// TwinCAT 3 PLC project vgr
// ProgramVersion: 3.1.4023.0
// libraries:
//   Tc2_Standard, * (Beckhoff Automation GmbH)
//   Tc2_System, * (Beckhoff Automation GmbH)
//   Tc3_Module, * (Beckhoff Automation GmbH)
// project tree:
//   GVLs/ Encoder.TcGVL, Position.TcGVL, StartStop.TcGVL, VGR.TcGVL
//   / PlcTask.TcTTO
//   POUs/ AboutEqual.TcPOU, AxisMovementController.TcPOU, AxisReferencing.TcPOU, EncoderSignalProcessor.TcPOU, MAIN.TcPOU, AxisController.TcPOU, VGR_State.TcPOU
// real-time tasks:
//   TASK PlcTask: cycle T#10ms, priority 20, ADS port 350
// I/O:
//   DEVICE Device 1 (EtherCAT), AmsNetId 172.23.144.1.2.1
//     Term 1 (EK1100) [EK1100 EtherCAT Coupler (2A E-Bus)]
//       Term 2 (EL1809) [EL1809 16Ch. Dig. Input 24V, 3ms]
//       Term 3 (EL2809) [EL2809 16Ch. Dig. Output 24V, 0.5A]
//       Term 4 (EL2535-0002) [EL2535-0002 2Ch. Pulse Width Current Output (24V, 2 A)]
//       Term 5 (EL2535-0002) [EL2535-0002 2Ch. Pulse Width Current Output (24V, 2 A)]
//       Term 6 (EL5152) [EL5152 2Ch. Inc. Encoder]
//       Term 7 (EL5152) [EL5152 2Ch. Inc. Encoder]
//       Term 8 (EL9011) [EL9011 End Terminal]
// variable links:
//   vgr/vgr Instance <-> Device 1 (EtherCAT)/Term 1 (EK1100)/Term 2 (EL1809)
//     PlcTask Inputs/StartStop.IX_START <-> Channel 11/Input
//     PlcTask Inputs/StartStop.IX_STOP <-> Channel 10/Input
//     PlcTask Inputs/VGR.IX_VGR_RefSwitchHorizontalAxis_I2 <-> Channel 2/Input
//     PlcTask Inputs/VGR.IX_VGR_RefSwitchRotate_I3 <-> Channel 3/Input
//     PlcTask Inputs/VGR.IX_VGR_RefSwitchVerticalAxis_I1 <-> Channel 1/Input
//   vgr/vgr Instance <-> Device 1 (EtherCAT)/Term 1 (EK1100)/Term 3 (EL2809)
//     PlcTask Outputs/VGR.QX_VGR_Compressor_Q7 <-> Channel 7/Output
//     PlcTask Outputs/VGR.QX_VGR_M1_VerticalAxisDown_Q2 <-> Channel 2/Output
//     PlcTask Outputs/VGR.QX_VGR_M1_VerticalAxisUp_Q1 <-> Channel 1/Output
//     PlcTask Outputs/VGR.QX_VGR_M2_HorizontalAxisBackward_Q3 <-> Channel 3/Output
//     PlcTask Outputs/VGR.QX_VGR_M2_HorizontalAxisForward_Q4 <-> Channel 4/Output
//     PlcTask Outputs/VGR.QX_VGR_M3_RotateClockwise_Q5 <-> Channel 5/Output
//     PlcTask Outputs/VGR.QX_VGR_M3_RotateCounterclockwise_Q6 <-> Channel 6/Output
//     PlcTask Outputs/VGR.QX_VGR_ValveVacuum_Q8 <-> Channel 8/Output
//   vgr/vgr Instance <-> Device 1 (EtherCAT)/Term 1 (EK1100)/Term 4 (EL2535-0002)
//     PlcTask Outputs/VGR.QW_VGR_PWM_Horizontal_Control <-> PWM Control Channel 2/Control
//     PlcTask Outputs/VGR.QW_VGR_PWM_Horizontal_M2 <-> PWM Control Channel 2/PWM output
//     PlcTask Outputs/VGR.QW_VGR_PWM_Vertical_Control <-> PWM Control Channel 1/Control
//     PlcTask Outputs/VGR.QW_VGR_PWM_Vertical_M1 <-> PWM Control Channel 1/PWM output
//   vgr/vgr Instance <-> Device 1 (EtherCAT)/Term 1 (EK1100)/Term 5 (EL2535-0002)
//     PlcTask Outputs/VGR.QW_VGR_PWM_Rotate_Control <-> PWM Control Channel 1/Control
//     PlcTask Outputs/VGR.QW_VGR_PWM_Rotate_M3 <-> PWM Control Channel 1/PWM output
//   vgr/vgr Instance <-> Device 1 (EtherCAT)/Term 1 (EK1100)/Term 6 (EL5152)
//     PlcTask Inputs/Encoder.countEncoderHorizontal <-> ENC Status compact Channel 2/Counter value
//     PlcTask Inputs/Encoder.countEncoderVertical <-> ENC Status compact Channel 1/Counter value
//     PlcTask Inputs/VGR.IX_VGR_EncoderHorizontalAxisImp1_B3 <-> ENC Status compact Channel 2/Status/Status of input A
//     PlcTask Inputs/VGR.IX_VGR_EncoderHorizontalAxisImp2_B4 <-> ENC Status compact Channel 2/Status/Status of input B
//     PlcTask Inputs/VGR.IX_VGR_EncoderVerticalAxisImp1_B1 <-> ENC Status compact Channel 1/Status/Status of input A
//     PlcTask Inputs/VGR.IX_VGR_EncoderVerticalAxisImp2_B2 <-> ENC Status compact Channel 1/Status/Status of input B
//     PlcTask Outputs/Encoder.setCounterHorizontal <-> ENC Control compact Channel 2/Control/Set counter
//     PlcTask Outputs/Encoder.setCounterValueHorizontal <-> ENC Control compact Channel 2/Set counter value
//     PlcTask Outputs/Encoder.setCounterValueVertical <-> ENC Control compact Channel 1/Set counter value
//     PlcTask Outputs/Encoder.setCounterVertical <-> ENC Control compact Channel 1/Control/Set counter
//   vgr/vgr Instance <-> Device 1 (EtherCAT)/Term 1 (EK1100)/Term 7 (EL5152)
//     PlcTask Inputs/Encoder.countEncoderRotate <-> ENC Status compact Channel 1/Counter value
//     PlcTask Inputs/VGR.IX_VGR_EncoderRotateImp1_B5 <-> ENC Status compact Channel 1/Status/Status of input A
//     PlcTask Inputs/VGR.IX_VGR_EncoderRotateImp2_B6 <-> ENC Status compact Channel 1/Status/Status of input B
//     PlcTask Outputs/Encoder.setCounterRotate <-> ENC Control compact Channel 1/Control/Set counter
//     PlcTask Outputs/Encoder.setCounterValueRotate <-> ENC Control compact Channel 1/Set counter value

CONFIGURATION vgr
    RESOURCE PLC ON TwinCAT3
        TASK PlcTask(INTERVAL := T#10ms, PRIORITY := 20);
        PROGRAM MAIN WITH PlcTask : MAIN;
    END_RESOURCE
END_CONFIGURATION

// ---- GVLs/Encoder.TcGVL
{attribute 'qualified_only'}
VAR_GLOBAL
	countEncoderVertical  AT %I* : UINT;
	countEncoderHorizontal  AT %I* : UINT;
	countEncoderRotate  AT %I* : UINT;
	setCounterValueVertical AT %Q* : UINT := 0;
	setCounterVertical AT %Q* : BOOL;
	setCounterValueHorizontal AT %Q* : UINT := 0;
	setCounterHorizontal AT %Q* : BOOL;
	setCounterValueRotate AT %Q* : UINT := 0;
	setCounterRotate AT %Q* : BOOL;
	
END_VAR

// ---- GVLs/Position.TcGVL
{attribute 'qualified_only'}
VAR_GLOBAL
	pickPositionVertical : UINT := 500;
	pickPositionHorizontal : UINT := 500;
	pickPositionRotation : UINT := 500;
	placePositionVertical : UINT := 100;
	placePositionHorizontal : UINT := 100;
	placePositionRotation : UINT := 200;
END_VAR

// ---- GVLs/StartStop.TcGVL
{attribute 'qualified_only'}
VAR_GLOBAL

IX_START AT %I*: BOOL;
IX_STOP AT %I*:	BOOL;
	
END_VAR

// ---- GVLs/VGR.TcGVL
{attribute 'qualified_only'}
VAR_GLOBAL

IX_VGR_RefSwitchVerticalAxis_I1 AT %I*: BOOL; //VGR - I1 = Reference switch vertical axis
IX_VGR_RefSwitchHorizontalAxis_I2 AT %I*: BOOL;//VGR - I2 = Reference switch horizontal axis
IX_VGR_RefSwitchRotate_I3 AT %I*: BOOL; //VGR - I3 = Reference switch rotate      
IX_VGR_EncoderVerticalAxisImp1_B1 AT %I* : BOOL; //VGR - Vertical axis encoder - Channel A
IX_VGR_EncoderVerticalAxisImp2_B2 AT %I* : BOOL; //VGR - Vertical axis encoder - Channel B
IX_VGR_EncoderHorizontalAxisImp1_B3 AT %I* : BOOL; //VGR - Horizontal axis encoder - Channel A
IX_VGR_EncoderHorizontalAxisImp2_B4 AT %I* : BOOL; //VGR - Horizontal axis encoder - Channel B
IX_VGR_EncoderRotateImp1_B5 AT %I* : BOOL; //VGR - Rotational axis encoder - Channel A
IX_VGR_EncoderRotateImp2_B6 AT %I* : BOOL; //VGR - Rotational axis encoder - Channel B
QX_VGR_M1_VerticalAxisUp_Q1 AT %Q* : BOOL; //VGR - Q1 = Motor M1 vertical axis up
QX_VGR_M1_VerticalAxisDown_Q2 AT %Q* : BOOL; //VGR - Q2 = Motor M1 vertical axis down
QX_VGR_M2_HorizontalAxisBackward_Q3 AT %Q* : BOOL; //VGR - Q3 = Motor M2 horizontal axis backward
QX_VGR_M2_HorizontalAxisForward_Q4 AT %Q* : BOOL; //VGR - Q4 = Motor M2 horizontal axis forward
QX_VGR_M3_RotateClockwise_Q5 AT %Q* : BOOL; //VGR - Q5 = Motor M3 rotate clockwise
QX_VGR_M3_RotateCounterclockwise_Q6 AT %Q* : BOOL; //VGR - Q6 = Motor M3 rotate counterclockwise
QX_VGR_Compressor_Q7 AT %Q* : BOOL; //VGR - Q7 = Compressor
QX_VGR_ValveVacuum_Q8 AT %Q* : BOOL; //VGR - Q8 = Valve vacuum
QW_VGR_PWM_Vertical_Control AT %Q* : INT; //VGR = PWM Motor M1 vertical axis enable
QW_VGR_PWM_Vertical_M1 AT %Q* : INT; //VGR = PWM Motor M1 vertical axis
QW_VGR_PWM_Horizontal_Control AT %Q* : INT; //VGR = PWM Motor M2 horizontal axis enable
QW_VGR_PWM_Horizontal_M2 AT %Q* : INT; //VGR = PWM Motor M2 horizontal axis
QW_VGR_PWM_Rotate_Control AT %Q* : INT; //VGR = PWM Motor M3 rotate axis enable
QW_VGR_PWM_Rotate_M3 AT %Q* : INT; //VGR = PWM Motor M3 rotate axis 	
END_VAR

// ---- POUs/MAIN.TcPOU
PROGRAM MAIN
VAR
	
END_VAR


Encoder.setCounterHorizontal := FALSE;
Encoder.setCounterRotate := FALSE;
Encoder.setCounterVertical := FALSE;

VGR_State();
(*
IF StartStop.IX_START THEN
VGR.QW_VGR_PWM_Vertical_Control := 32;
VGR.QW_VGR_PWM_Vertical_M1 := 3000;
VGR.QX_VGR_M1_VerticalAxisDown_Q2 := TRUE;
ELSIF NOT StartStop.IX_STOP THEN
VGR.QW_VGR_PWM_Vertical_Control := 32;
VGR.QW_VGR_PWM_Vertical_M1 := 3000;
VGR.QX_VGR_M1_VerticalAxisUp_Q1 := TRUE;
ELSE
	VGR.QX_VGR_M1_VerticalAxisUp_Q1 := FALSE;
	VGR.QX_VGR_M1_VerticalAxisDown_Q2 := FALSE;
	VGR.QW_VGR_PWM_Vertical_Control := 0;
VGR.QW_VGR_PWM_Vertical_M1 := 0;
END_IF
*)

END_PROGRAM

// ---- POUs/VGR_State.TcPOU
PROGRAM VGR_State
VAR
	
	bStateIdle: BOOL := TRUE;
	bStatePlace: BOOL;
	bStateHoming: BOOL;
	bStatePick: BOOL;
	tolerance : UINT := 5;
	
	bInPositionPickVertical : BOOL;
	bInPositionPickHorizontal : BOOL;
	bInPositionPickRotate : BOOL;
	bInPositionPlaceVertical : BOOL;
	bInPositionPlaceHorizontal : BOOL;
	bInPositionPlaceRotate : BOOL;
	
	bValveClosed : BOOL;
	
	RS_Idle: RS;
	
	RS_Homing: RS;
	
	RS_Pick: RS;
	bValveOpened: BOOL;
	RS_Place: RS;
	bValveOpen: BOOL;
	SR_ESTOP: SR;
	bStateEStop: BOOL;
	AxisMovementController_Vertical: AxisMovementController;
	AxisMovementController_Horizontal: AxisMovementController;
	AxisReferencing_Vertical: AxisReferencing;
	AxisReferencing_Horizontal: AxisReferencing;
	AxisReferencing_Rotational: AxisReferencing;
	AxisMovementController_Rotation: AxisMovementController;
END_VAR
VAR // added by the converter: edge detectors and wires of the graphical bodies
    _w1 : BOOL;
END_VAR

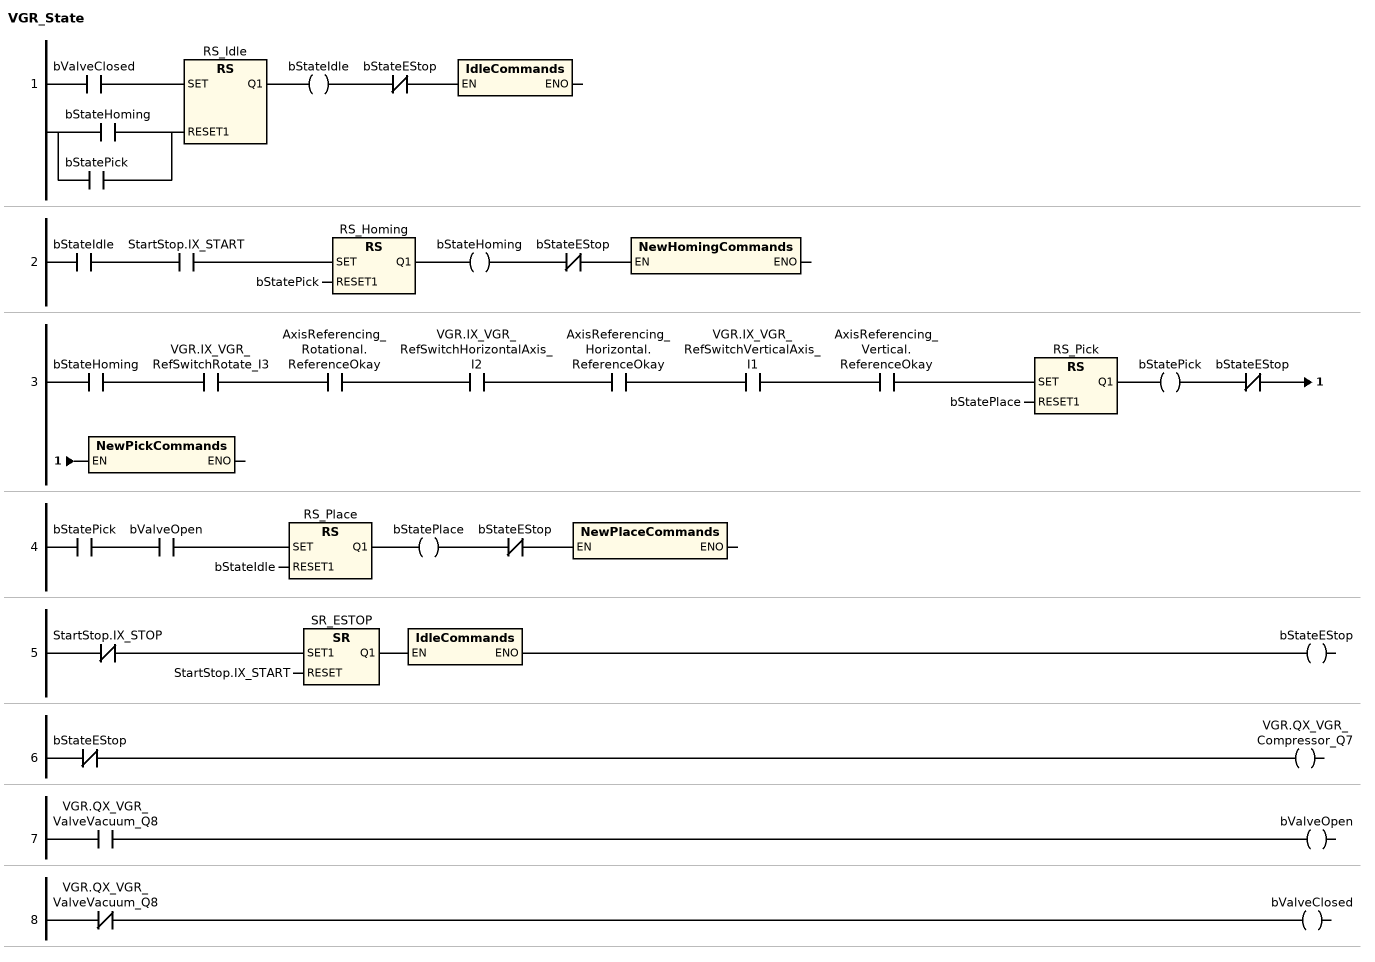
// NETWORK 1
RS_Idle(SET := bValveClosed, RESET1 := bStateHoming OR bStatePick); // RS
bStateIdle := RS_Idle.Q1;
IF RS_Idle.Q1 AND NOT bStateEStop THEN IdleCommands(); END_IF

// NETWORK 2
RS_Homing(SET := bStateIdle AND StartStop.IX_START, RESET1 := bStatePick); // RS
bStateHoming := RS_Homing.Q1;
IF RS_Homing.Q1 AND NOT bStateEStop THEN NewHomingCommands(); END_IF

// NETWORK 3
RS_Pick(SET := bStateHoming AND VGR.IX_VGR_RefSwitchRotate_I3 AND AxisReferencing_Rotational.ReferenceOkay AND VGR.IX_VGR_RefSwitchHorizontalAxis_I2 AND AxisReferencing_Horizontal.ReferenceOkay AND VGR.IX_VGR_RefSwitchVerticalAxis_I1 AND AxisReferencing_Vertical.ReferenceOkay, RESET1 := bStatePlace); // RS
bStatePick := RS_Pick.Q1;
IF RS_Pick.Q1 AND NOT bStateEStop THEN NewPickCommands(); END_IF

// NETWORK 4
RS_Place(SET := bStatePick AND bValveOpen, RESET1 := bStateIdle); // RS
bStatePlace := RS_Place.Q1;
IF RS_Place.Q1 AND NOT bStateEStop THEN NewPlaceCommands(); END_IF

// NETWORK 5
SR_ESTOP(SET1 := NOT StartStop.IX_STOP, RESET := StartStop.IX_START); // SR
_w1 := SR_ESTOP.Q1;
IF _w1 THEN IdleCommands(); END_IF
bStateEStop := _w1;

// NETWORK 6
VGR.QX_VGR_Compressor_Q7 := NOT bStateEStop;

// NETWORK 7
bValveOpen := VGR.QX_VGR_ValveVacuum_Q8;

// NETWORK 8
bValveClosed := NOT VGR.QX_VGR_ValveVacuum_Q8;

ACTION HomeCommands:
IF VGR.IX_VGR_RefSwitchVerticalAxis_I1 THEN
	VGR.QX_VGR_M1_VerticalAxisUp_Q1 := FALSE;
	VGR.QX_VGR_M1_VerticalAxisDown_Q2 := FALSE;
	VGR.QW_VGR_PWM_Vertical_Control := 0;
	VGR.QW_VGR_PWM_Vertical_M1 := 0;
	Encoder.setCounterVertical := TRUE;
	Encoder.setCounterValueVertical:= 0;
ELSE
	VGR.QX_VGR_M1_VerticalAxisUp_Q1 := TRUE;
	VGR.QX_VGR_M1_VerticalAxisDown_Q2 := FALSE;
	VGR.QW_VGR_PWM_Vertical_Control := 32;
	VGR.QW_VGR_PWM_Vertical_M1 := 5000;
END_IF
IF VGR.IX_VGR_RefSwitchHorizontalAxis_I2 THEN
	VGR.QX_VGR_M2_HorizontalAxisBackward_Q3 := FALSE;
    VGR.QX_VGR_M2_HorizontalAxisForward_Q4 := FALSE;
    VGR.QW_VGR_PWM_Horizontal_Control := 0;
    VGR.QW_VGR_PWM_Horizontal_M2 := 0;
	Encoder.setCounterHorizontal := TRUE;
ELSE
	VGR.QX_VGR_M2_HorizontalAxisBackward_Q3 := TRUE;
    VGR.QX_VGR_M2_HorizontalAxisForward_Q4 := FALSE;
    VGR.QW_VGR_PWM_Horizontal_Control := 32;
    VGR.QW_VGR_PWM_Horizontal_M2 := 5000;
END_IF
IF VGR.IX_VGR_RefSwitchHorizontalAxis_I2 THEN
	VGR.QX_VGR_M3_RotateClockwise_Q5 := FALSE;
    VGR.QX_VGR_M3_RotateCounterClockwise_Q6 := FALSE;
    VGR.QW_VGR_PWM_Rotate_Control := 0;
    VGR.QW_VGR_PWM_Rotate_M3 := 0;
	Encoder.setCounterRotate := TRUE;
ELSE
	VGR.QX_VGR_M3_RotateClockwise_Q5 := TRUE;
    VGR.QX_VGR_M3_RotateCounterClockwise_Q6 := FALSE;
    VGR.QW_VGR_PWM_Rotate_Control := 32;
    VGR.QW_VGR_PWM_Rotate_M3 := 5000;
END_IF
END_ACTION

ACTION IdleCommands:
VGR.QX_VGR_M1_VerticalAxisUp_Q1 := FALSE;
VGR.QX_VGR_M1_VerticalAxisDown_Q2 := FALSE;
VGR.QW_VGR_PWM_Vertical_Control := 0;
VGR.QW_VGR_PWM_Vertical_M1 := 0;
VGR.QX_VGR_M2_HorizontalAxisBackward_Q3 := FALSE;
VGR.QX_VGR_M2_HorizontalAxisForward_Q4 := FALSE;
VGR.QW_VGR_PWM_Horizontal_Control := 0;
VGR.QW_VGR_PWM_Horizontal_M2 := 0;
VGR.QX_VGR_M3_RotateClockwise_Q5 := FALSE;
VGR.QX_VGR_M3_RotateCounterClockwise_Q6 := FALSE;
VGR.QW_VGR_PWM_Rotate_Control := 0;
VGR.QW_VGR_PWM_Rotate_M3 := 0;
END_ACTION

ACTION NewHomingCommands:
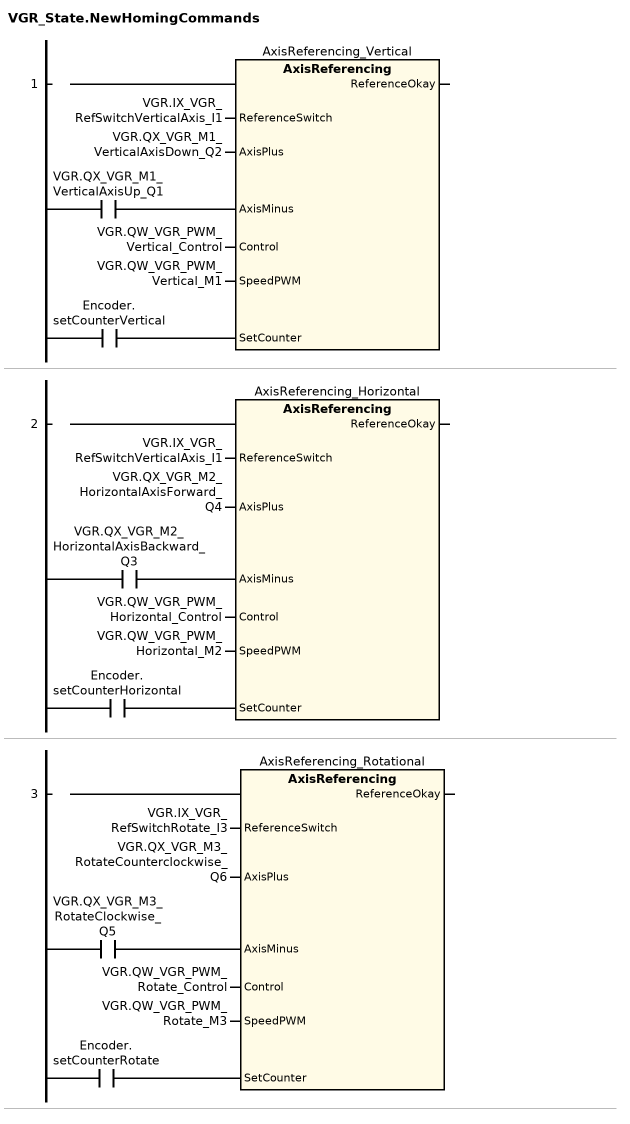
// NETWORK 1
AxisReferencing_Vertical(
    ReferenceSwitch := VGR.IX_VGR_RefSwitchVerticalAxis_I1,
    AxisPlus := VGR.QX_VGR_M1_VerticalAxisDown_Q2,
    AxisMinus := VGR.QX_VGR_M1_VerticalAxisUp_Q1,
    Control := VGR.QW_VGR_PWM_Vertical_Control,
    SpeedPWM := VGR.QW_VGR_PWM_Vertical_M1,
    SetCounter := Encoder.setCounterVertical); // AxisReferencing

// NETWORK 2
AxisReferencing_Horizontal(
    ReferenceSwitch := VGR.IX_VGR_RefSwitchVerticalAxis_I1,
    AxisPlus := VGR.QX_VGR_M2_HorizontalAxisForward_Q4,
    AxisMinus := VGR.QX_VGR_M2_HorizontalAxisBackward_Q3,
    Control := VGR.QW_VGR_PWM_Horizontal_Control,
    SpeedPWM := VGR.QW_VGR_PWM_Horizontal_M2,
    SetCounter := Encoder.setCounterHorizontal); // AxisReferencing

// NETWORK 3
AxisReferencing_Rotational(
    ReferenceSwitch := VGR.IX_VGR_RefSwitchRotate_I3,
    AxisPlus := VGR.QX_VGR_M3_RotateCounterclockwise_Q6,
    AxisMinus := VGR.QX_VGR_M3_RotateClockwise_Q5,
    Control := VGR.QW_VGR_PWM_Rotate_Control,
    SpeedPWM := VGR.QW_VGR_PWM_Rotate_M3,
    SetCounter := Encoder.setCounterRotate); // AxisReferencing
END_ACTION

ACTION NewPickCommands:
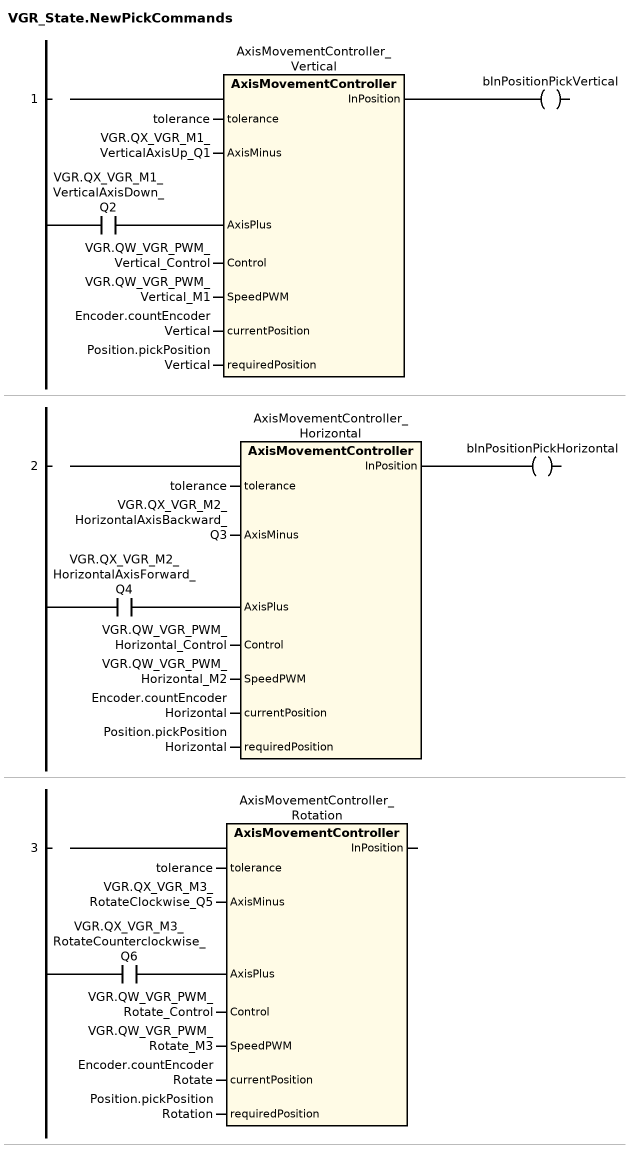
// NETWORK 1
AxisMovementController_Vertical(
    tolerance := tolerance,
    AxisMinus := VGR.QX_VGR_M1_VerticalAxisUp_Q1,
    AxisPlus := VGR.QX_VGR_M1_VerticalAxisDown_Q2,
    Control := VGR.QW_VGR_PWM_Vertical_Control,
    SpeedPWM := VGR.QW_VGR_PWM_Vertical_M1,
    currentPosition := Encoder.countEncoderVertical,
    requiredPosition := Position.pickPositionVertical); // AxisMovementController
bInPositionPickVertical := AxisMovementController_Vertical.InPosition;

// NETWORK 2
AxisMovementController_Horizontal(
    tolerance := tolerance,
    AxisMinus := VGR.QX_VGR_M2_HorizontalAxisBackward_Q3,
    AxisPlus := VGR.QX_VGR_M2_HorizontalAxisForward_Q4,
    Control := VGR.QW_VGR_PWM_Horizontal_Control,
    SpeedPWM := VGR.QW_VGR_PWM_Horizontal_M2,
    currentPosition := Encoder.countEncoderHorizontal,
    requiredPosition := Position.pickPositionHorizontal); // AxisMovementController
bInPositionPickHorizontal := AxisMovementController_Horizontal.InPosition;

// NETWORK 3
AxisMovementController_Rotation(
    tolerance := tolerance,
    AxisMinus := VGR.QX_VGR_M3_RotateClockwise_Q5,
    AxisPlus := VGR.QX_VGR_M3_RotateCounterclockwise_Q6,
    Control := VGR.QW_VGR_PWM_Rotate_Control,
    SpeedPWM := VGR.QW_VGR_PWM_Rotate_M3,
    currentPosition := Encoder.countEncoderRotate,
    requiredPosition := Position.pickPositionRotation); // AxisMovementController
END_ACTION

ACTION NewPlaceCommands:
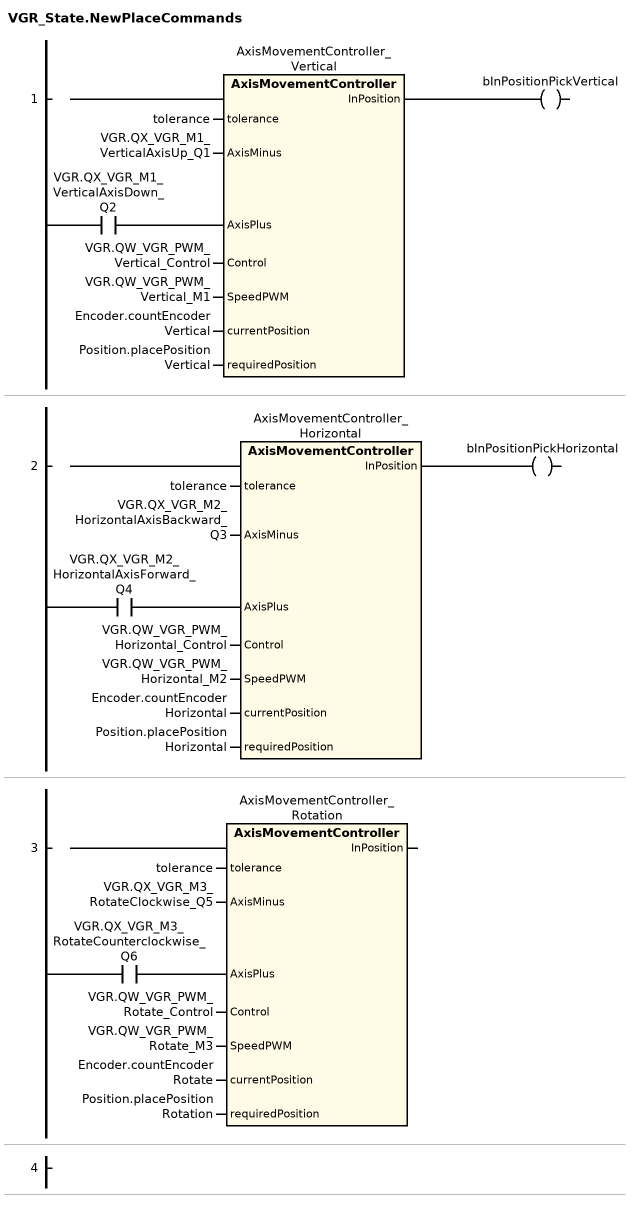
// NETWORK 1
AxisMovementController_Vertical(
    tolerance := tolerance,
    AxisMinus := VGR.QX_VGR_M1_VerticalAxisUp_Q1,
    AxisPlus := VGR.QX_VGR_M1_VerticalAxisDown_Q2,
    Control := VGR.QW_VGR_PWM_Vertical_Control,
    SpeedPWM := VGR.QW_VGR_PWM_Vertical_M1,
    currentPosition := Encoder.countEncoderVertical,
    requiredPosition := Position.placePositionVertical); // AxisMovementController
bInPositionPickVertical := AxisMovementController_Vertical.InPosition;

// NETWORK 2
AxisMovementController_Horizontal(
    tolerance := tolerance,
    AxisMinus := VGR.QX_VGR_M2_HorizontalAxisBackward_Q3,
    AxisPlus := VGR.QX_VGR_M2_HorizontalAxisForward_Q4,
    Control := VGR.QW_VGR_PWM_Horizontal_Control,
    SpeedPWM := VGR.QW_VGR_PWM_Horizontal_M2,
    currentPosition := Encoder.countEncoderHorizontal,
    requiredPosition := Position.placePositionHorizontal); // AxisMovementController
bInPositionPickHorizontal := AxisMovementController_Horizontal.InPosition;

// NETWORK 3
AxisMovementController_Rotation(
    tolerance := tolerance,
    AxisMinus := VGR.QX_VGR_M3_RotateClockwise_Q5,
    AxisPlus := VGR.QX_VGR_M3_RotateCounterclockwise_Q6,
    Control := VGR.QW_VGR_PWM_Rotate_Control,
    SpeedPWM := VGR.QW_VGR_PWM_Rotate_M3,
    currentPosition := Encoder.countEncoderRotate,
    requiredPosition := Position.placePositionRotation); // AxisMovementController

// NETWORK 4
END_ACTION

ACTION PickCommands:
IF  AboutEqual(IN1:= Encoder.countEncoderVertical,
	IN2:= Position.pickPositionVertical,
Tolerance:= tolerance)
 THEN
	VGR.QX_VGR_M1_VerticalAxisUp_Q1 := FALSE;
	VGR.QX_VGR_M1_VerticalAxisDown_Q2 := FALSE;
	VGR.QW_VGR_PWM_Vertical_Control := 0;
	VGR.QW_VGR_PWM_Vertical_M1 := 0;
	bInPositionPickVertical := TRUE;
ELSIF Encoder.countEncoderVertical > Position.pickPositionVertical AND NOT bInPositionPickVertical THEN
	VGR.QX_VGR_M1_VerticalAxisUp_Q1 := TRUE;
	VGR.QX_VGR_M1_VerticalAxisDown_Q2 := FALSE;
	VGR.QW_VGR_PWM_Vertical_Control := 32;
	VGR.QW_VGR_PWM_Vertical_M1 := 5000;
	bInPositionPickVertical := FALSE;
ELSE
	VGR.QX_VGR_M1_VerticalAxisUp_Q1 := FALSE;
	VGR.QX_VGR_M1_VerticalAxisDown_Q2 := TRUE;
	VGR.QW_VGR_PWM_Vertical_Control := 32;
	VGR.QW_VGR_PWM_Vertical_M1 := 5000;
	bInPositionPickVertical := FALSE;
END_IF
IF AboutEqual(IN1:= Encoder.countEncoderHorizontal,
	IN2:= Position.pickPositionHorizontal,
Tolerance:= tolerance) THEN
	VGR.QX_VGR_M2_HorizontalAxisBackward_Q3 := FALSE;
    VGR.QX_VGR_M2_HorizontalAxisForward_Q4 := FALSE;
    VGR.QW_VGR_PWM_Horizontal_Control := 0;
    VGR.QW_VGR_PWM_Horizontal_M2 := 0;
	bInPositionPickHorizontal := TRUE;
ELSIF Encoder.countEncoderHorizontal > Position.pickPositionHorizontal  AND NOT bInPositionPickHorizontal THEN
	VGR.QX_VGR_M2_HorizontalAxisBackward_Q3 := TRUE;
    VGR.QX_VGR_M2_HorizontalAxisForward_Q4 := FALSE;
    VGR.QW_VGR_PWM_Horizontal_Control := 32;
    VGR.QW_VGR_PWM_Horizontal_M2 := 5000;
	bInPositionPickHorizontal := FALSE;
ELSE
	VGR.QX_VGR_M2_HorizontalAxisBackward_Q3 := FALSE;
	VGR.QX_VGR_M2_HorizontalAxisForward_Q4 := TRUE;
	VGR.QW_VGR_PWM_Horizontal_Control := 32;
	VGR.QW_VGR_PWM_Horizontal_M2 := 5000;
	bInPositionPickHorizontal := FALSE;
END_IF
IF  AboutEqual(IN1:= Encoder.countEncoderRotate,
	IN2:= Position.pickPositionRotation,
Tolerance:= tolerance) THEN
    VGR.QX_VGR_M3_RotateClockwise_Q5 := FALSE;
    VGR.QX_VGR_M3_RotateCounterClockwise_Q6 := FALSE;
    VGR.QW_VGR_PWM_Rotate_Control := 0;
    VGR.QW_VGR_PWM_Rotate_M3 := 0;
	bInPositionPickRotate := TRUE;
ELSIF Encoder.countEncoderRotate > Position.pickPositionRotation  AND NOT bInPositionPickRotate THEN
	VGR.QX_VGR_M3_RotateClockwise_Q5 := FALSE;
    VGR.QX_VGR_M3_RotateCounterClockwise_Q6 := TRUE;
    VGR.QW_VGR_PWM_Rotate_Control := 32;
    VGR.QW_VGR_PWM_Rotate_M3 := 5000;
	bInPositionPickRotate := FALSE;
ELSE
	VGR.QX_VGR_M3_RotateClockwise_Q5 := TRUE;
    VGR.QX_VGR_M3_RotateCounterClockwise_Q6 := FALSE;
    VGR.QW_VGR_PWM_Rotate_Control := 32;
    VGR.QW_VGR_PWM_Rotate_M3 := 5000;
	bInPositionPickRotate := FALSE;
END_IF

IF bInPositionPickRotate AND bInPositionPickRotate AND bInPositionPickRotate THEN
	VGR.QX_VGR_ValveVacuum_Q8 := TRUE;
ELSE
	VGR.QX_VGR_ValveVacuum_Q8 := FALSE;
END_IF
END_ACTION

ACTION PlaceCommands:
IF  Encoder.countEncoderVertical = Position.placePositionVertical OR
	(Position.pickPositionVertical+tolerance > Encoder.countEncoderVertical OR 
	Encoder.countEncoderVertical > Position.pickPositionVertical-tolerance ) THEN
	VGR.QX_VGR_M1_VerticalAxisUp_Q1 := FALSE;
	VGR.QX_VGR_M1_VerticalAxisDown_Q2 := FALSE;
	VGR.QW_VGR_PWM_Vertical_Control := 0;
	VGR.QW_VGR_PWM_Vertical_M1 := 0;
	bInPositionPlaceVertical := TRUE;
ELSIF Encoder.countEncoderVertical > Position.placePositionVertical THEN
	VGR.QX_VGR_M1_VerticalAxisUp_Q1 := FALSE;
	VGR.QX_VGR_M1_VerticalAxisDown_Q2 := TRUE;
	VGR.QW_VGR_PWM_Vertical_Control := 32;
	VGR.QW_VGR_PWM_Vertical_M1 := 5000;
	bInPositionPlaceVertical := FALSE;
ELSE
	VGR.QX_VGR_M1_VerticalAxisUp_Q1 := TRUE;
	VGR.QX_VGR_M1_VerticalAxisDown_Q2 := FALSE;
	VGR.QW_VGR_PWM_Vertical_Control := 32;
	VGR.QW_VGR_PWM_Vertical_M1 := 5000;
	bInPositionPlaceVertical := FALSE;
END_IF
IF Encoder.countEncoderHorizontal = Position.placePositionHorizontal OR 
(Encoder.countEncoderHorizontal < Position.pickPositionHorizontal + tolerance)OR 
(Encoder.countEncoderHorizontal > Position.pickPositionHorizontal -tolerance) THEN
	VGR.QX_VGR_M2_HorizontalAxisBackward_Q3 := FALSE;
    VGR.QX_VGR_M2_HorizontalAxisForward_Q4 := FALSE;
    VGR.QW_VGR_PWM_Horizontal_Control := 0;
    VGR.QW_VGR_PWM_Horizontal_M2 := 0;
	bInPositionPlaceHorizontal := TRUE;
ELSIF Encoder.countEncoderHorizontal > Position.placePositionHorizontal THEN
	VGR.QX_VGR_M2_HorizontalAxisBackward_Q3 := TRUE;
    VGR.QX_VGR_M2_HorizontalAxisForward_Q4 := FALSE;
    VGR.QW_VGR_PWM_Horizontal_Control := 32;
    VGR.QW_VGR_PWM_Horizontal_M2 := 5000;
	bInPositionPlaceHorizontal := FALSE;
ELSE
	VGR.QX_VGR_M2_HorizontalAxisBackward_Q3 := FALSE;
	VGR.QX_VGR_M2_HorizontalAxisForward_Q4 := TRUE;
	VGR.QW_VGR_PWM_Horizontal_Control := 32;
	VGR.QW_VGR_PWM_Horizontal_M2 := 5000;
	bInPositionPlaceHorizontal := FALSE;
END_IF
IF  Encoder.countEncoderRotate=Position.placePositionRotation  OR 
(Encoder.countEncoderRotate < Position.pickPositionRotation+tolerance) OR 
(Encoder.countEncoderRotate>Position.pickPositionRotation-tolerance) THEN
    VGR.QX_VGR_M3_RotateClockwise_Q5 := FALSE;
    VGR.QX_VGR_M3_RotateCounterClockwise_Q6 := FALSE;
    VGR.QW_VGR_PWM_Rotate_Control := 0;
    VGR.QW_VGR_PWM_Rotate_M3 := 0;
	bInPositionPlaceRotate := TRUE;
ELSIF Encoder.countEncoderRotate > Position.placePositionRotation THEN
	VGR.QX_VGR_M3_RotateClockwise_Q5 := FALSE;
    VGR.QX_VGR_M3_RotateCounterClockwise_Q6 := TRUE;
    VGR.QW_VGR_PWM_Rotate_Control := 32;
    VGR.QW_VGR_PWM_Rotate_M3 := 5000;
	bInPositionPlaceRotate := FALSE;
ELSE
	VGR.QX_VGR_M3_RotateClockwise_Q5 := TRUE;
    VGR.QX_VGR_M3_RotateCounterClockwise_Q6 := FALSE;
    VGR.QW_VGR_PWM_Rotate_Control := 32;
    VGR.QW_VGR_PWM_Rotate_M3 := 5000;
	bInPositionPlaceRotate := FALSE;
END_IF

IF bInPositionPlaceHorizontal AND bInPositionPlaceRotate AND bInPositionPlaceVertical THEN
	VGR.QX_VGR_ValveVacuum_Q8 := FALSE;
ELSE
	VGR.QX_VGR_ValveVacuum_Q8 := TRUE;
END_IF
END_ACTION

END_PROGRAM

// ---- POUs/AxisMovementController.TcPOU
FUNCTION_BLOCK AxisMovementController
VAR_INPUT
	tolerance: UINT;
	AxisMinus : BOOL;
	AxisPlus: BOOL;
	Control: INT;
	SpeedPWM:INT;
	currentPosition : UINT;
	requiredPosition : UINT;
END_VAR
VAR_OUTPUT
	InPosition:BOOL;
END_VAR
VAR
END_VAR

IF  AboutEqual(
	IN1:= currentPosition,
	IN2:= requiredPosition,
	Tolerance:= tolerance
)
 THEN
	AxisMinus := FALSE;
	AxisPlus := FALSE;
	Control := 0;
	SpeedPWM := 0;
	InPosition := TRUE;
ELSIF currentPosition > requiredPosition AND NOT InPosition THEN
	AxisMinus := TRUE;
	AxisPlus := FALSE;
	Control:= 32;
	SpeedPWM := 5000;
	InPosition := FALSE;
ELSIF currentPosition < requiredPosition AND NOT InPosition THEN
	AxisMinus := FALSE;
	AxisPlus := TRUE;
	Control := 32;
	SpeedPWM := 5000;
	InPosition := FALSE;
ELSE
	AxisMinus := FALSE;
	AxisPlus := FALSE;
	Control := 0;
	SpeedPWM := 0;
	InPosition := FALSE;
END_IF

END_FUNCTION_BLOCK

// ---- POUs/AboutEqual.TcPOU
FUNCTION AboutEqual : BOOL
VAR_INPUT
	IN1: UINT;
	IN2: UINT;
	Tolerance: UINT;
END_VAR
VAR_OUTPUT
END_VAR
VAR
	Difference: UINT;
END_VAR

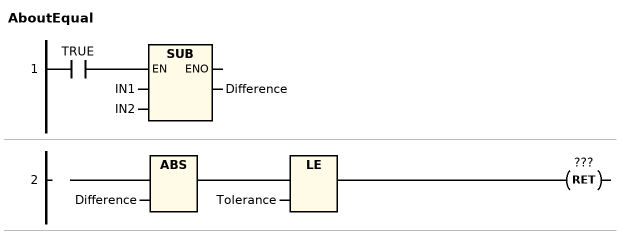
// NETWORK 1
Difference := IN1 - IN2;

// NETWORK 2
IF ABS(Difference) <= Tolerance THEN RETURN; END_IF

END_FUNCTION

// ---- POUs/AxisReferencing.TcPOU
FUNCTION_BLOCK AxisReferencing
VAR_IN_OUT
	ReferenceSwitch:BOOL;
	AxisPlus:BOOL;
	AxisMinus:BOOL;
	Control:INT;
	SpeedPWM:INT;
	SetCounter:BOOL;
END_VAR
VAR_OUTPUT
	ReferenceOkay:BOOL;
END_VAR
VAR
END_VAR

IF ReferenceSwitch THEN
	AxisMinus := FALSE;
	AxisPlus := FALSE;
	Control := 0;
	SpeedPWM := 0;
	SetCounter := TRUE;
	ReferenceOkay:= TRUE;
ELSE
	AxisMinus := TRUE;
	AxisPlus := FALSE;
	Control := 32;
	SpeedPWM := 5000;
	SetCounter := FALSE;
END_IF

END_FUNCTION_BLOCK

// ---- POUs/EncoderSignalProcessor.TcPOU
FUNCTION_BLOCK EncoderSignalProcessor
VAR_INPUT
	pulseA : BOOL;
	pulseB : BOOL;
	//reset :	
	referencePositionSensor : BOOL;
	referencePosition: INT := 0;
END_VAR
VAR_OUTPUT
	direction : BOOL;
	position : INT;
END_VAR
VAR
	trigger : BOOL;
	direction_ : BOOL;
	count_ : INT;
	
END_VAR
VAR // added by the converter: edge detectors and wires of the graphical bodies
    _rt1, _rt2, _rt3, _rt4 : R_TRIG;
    _ft1, _ft2, _ft3, _ft4 : F_TRIG;
END_VAR

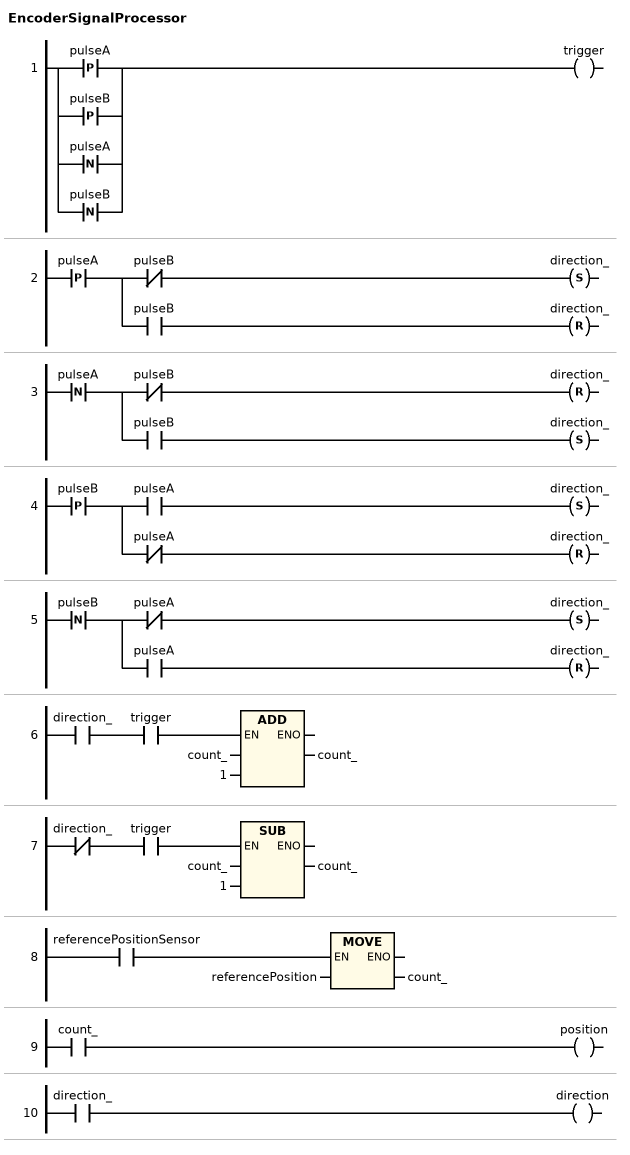
// NETWORK 1
_rt1(CLK := pulseA);
_rt2(CLK := pulseB);
_ft1(CLK := pulseA);
_ft2(CLK := pulseB);
trigger := _rt1.Q OR _rt2.Q OR _ft1.Q OR _ft2.Q;

// NETWORK 2
_rt3(CLK := pulseA);
direction_ S= _rt3.Q AND NOT pulseB;
direction_ R= _rt3.Q AND pulseB;

// NETWORK 3
_ft3(CLK := pulseA);
direction_ R= _ft3.Q AND NOT pulseB;
direction_ S= _ft3.Q AND pulseB;

// NETWORK 4
_rt4(CLK := pulseB);
direction_ S= _rt4.Q AND pulseA;
direction_ R= _rt4.Q AND NOT pulseA;

// NETWORK 5
_ft4(CLK := pulseB);
direction_ S= _ft4.Q AND NOT pulseA;
direction_ R= _ft4.Q AND pulseA;

// NETWORK 6
IF direction_ AND trigger THEN count_ := count_ + 1; END_IF

// NETWORK 7
IF NOT direction_ AND trigger THEN count_ := count_ - 1; END_IF

// NETWORK 8
IF referencePositionSensor THEN count_ := referencePosition; END_IF

// NETWORK 9
position := count_;

// NETWORK 10
direction := direction_;

END_FUNCTION_BLOCK

// ---- POUs/AxisController.TcPOU
PROGRAM AxisController
VAR
	directionVertical : BOOL;
	positionVertical : INT;
	EncoderSignalProcessor_Vertical: EncoderSignalProcessor;
	initialPosition: INT := 0;
	EncoderSignalProcessor_Horizontal: EncoderSignalProcessor;
	positionHorizontal: INT;
	directionHorizontal: BOOL;
	positionRotational: INT;
	directionRotational: BOOL;
	EncoderSignalProcessor_Rotational: EncoderSignalProcessor;
END_VAR

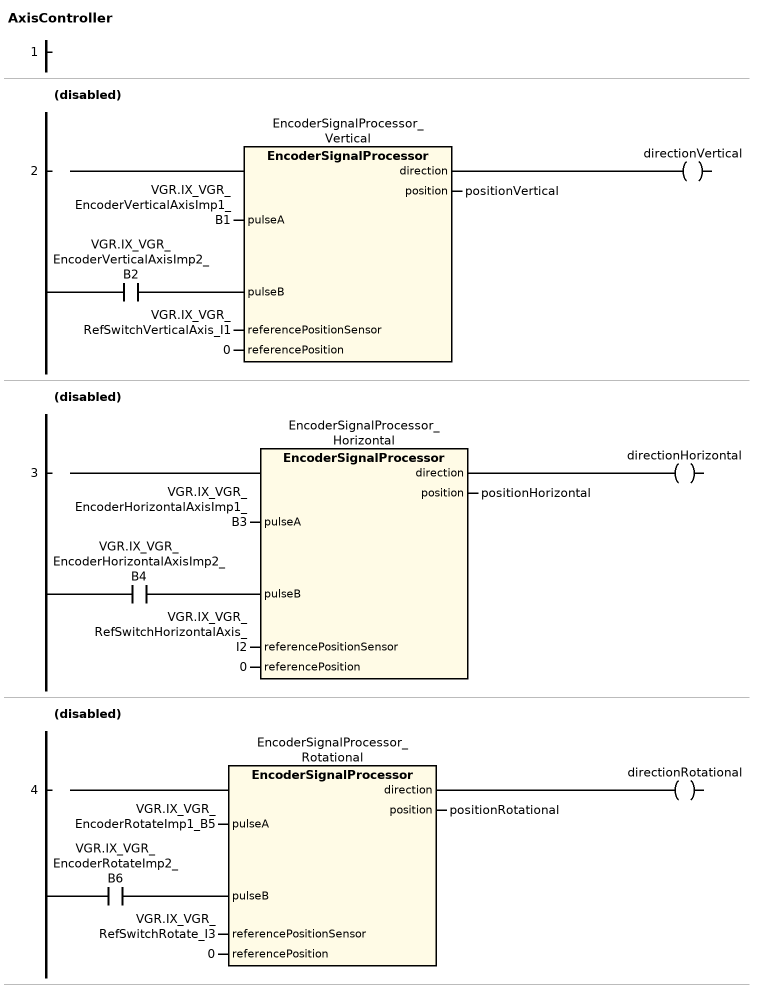
// NETWORK 1

// NETWORK 2 (disabled)
// EncoderSignalProcessor_Vertical(
//     pulseA := VGR.IX_VGR_EncoderVerticalAxisImp1_B1,
//     pulseB := VGR.IX_VGR_EncoderVerticalAxisImp2_B2,
//     referencePositionSensor := VGR.IX_VGR_RefSwitchVerticalAxis_I1,
//     referencePosition := 0,
//     position => positionVertical); // EncoderSignalProcessor
// directionVertical := EncoderSignalProcessor_Vertical.direction;

// NETWORK 3 (disabled)
// EncoderSignalProcessor_Horizontal(
//     pulseA := VGR.IX_VGR_EncoderHorizontalAxisImp1_B3,
//     pulseB := VGR.IX_VGR_EncoderHorizontalAxisImp2_B4,
//     referencePositionSensor := VGR.IX_VGR_RefSwitchHorizontalAxis_I2,
//     referencePosition := 0,
//     position => positionHorizontal); // EncoderSignalProcessor
// directionHorizontal := EncoderSignalProcessor_Horizontal.direction;

// NETWORK 4 (disabled)
// EncoderSignalProcessor_Rotational(
//     pulseA := VGR.IX_VGR_EncoderRotateImp1_B5,
//     pulseB := VGR.IX_VGR_EncoderRotateImp2_B6,
//     referencePositionSensor := VGR.IX_VGR_RefSwitchRotate_I3,
//     referencePosition := 0,
//     position => positionRotational); // EncoderSignalProcessor
// directionRotational := EncoderSignalProcessor_Rotational.direction;

END_PROGRAM
